RESOURCE_TYPE EMB_RES (* A Simple Embedded Resource Type *)
  (* Standard: 61499-1; Function: Device Management; Description: A simple embedded resource *)
  (* Version 0.1, 2007-10-10, JHC, Holobloc Inc, Moved to fb.rt. *)
  (* Version 0.0, 2001-01-04, JHC, Rockwell Automation *)
  (* Compiler header: package fb.rt; *)
  (* Compiler Java IBM VisualAge 3.0 *)
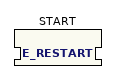
  FBS
    START : E_RESTART;
  END_FBS
END_RESOURCE_TYPE
